FUNCTION_BLOCK FB_BPFanout
VAR_INPUT

END_VAR
VAR_OUTPUT
    stBP    :    ST_BeamParams;
END_VAR
VAR
    i_stBP    AT %I* :    ST_BeamParams;
    
    xTxPDO_toggle    AT     %I* :    BIT;
    xTxPDO_state    AT    %I*    :    BIT;
END_VAR


stBP := i_stBP;
stBP.xValidToggle := xTxPDO_toggle;

PMPS_GVL.stCurrentBeamParameters := stBP;

END_FUNCTION_BLOCK

(* stored: Version 1.1.0.1, ProductVersion 3.1.4022.18
   POU FB_BPFanout: Id {46d56ca5-5404-4b6a-916e-f0dea48641e9}, SpecialFunc None *)
